SUBAPPLICATION Uebung_039_sub_Outputs (* Spiegelabfolge V2 mit Schrittkette SUB Out *)
  (* Standard: 61499-2 *)
  (* Version 1.0, 2024-03-03, franz *)
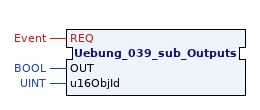
  EVENT_INPUT
    REQ; (* Service Request *)
  END_EVENT
  VAR_INPUT
    OUT : BOOL; (* Output data to resource *)
    u16ObjId : UINT := ID_NULL; (* Object ID Softkey/Button *)
  END_VAR
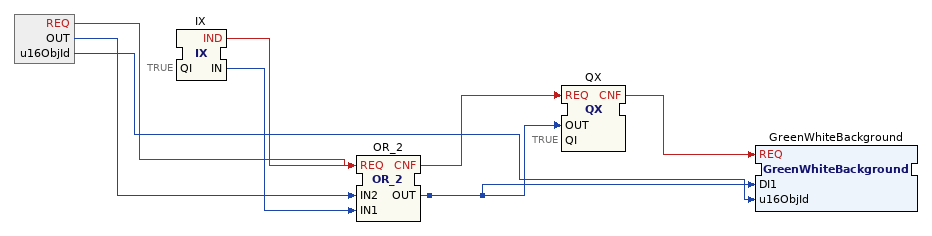
  FBS
    QX : QX(QI := TRUE);
    IX : IX(QI := TRUE);
    OR_2 : OR_2;
  END_FBS
  SUBAPPS
    GreenWhiteBackground : GreenWhiteBackground;
  END_SUBAPPS
  EVENT_CONNECTIONS
    OR_2.CNF TO QX.REQ;
    IX.IND TO OR_2.REQ;
    REQ TO OR_2.REQ;
    QX.CNF TO GreenWhiteBackground.REQ;
  END_CONNECTIONS
  DATA_CONNECTIONS
    OUT TO OR_2.IN2;
    IX.IN TO OR_2.IN1;
    OR_2.OUT TO QX.OUT;
    OR_2.OUT TO GreenWhiteBackground.DI1;
    u16ObjId TO GreenWhiteBackground.u16ObjId;
  END_CONNECTIONS
END_SUBAPPLICATION
